TYPE ST_HMI_Machine :
STRUCT
	Command: ST_HMI_Machine_Command;
	Config: ST_HMI_Machine_Config;
	Status: ST_HMI_Machine_Status;
END_STRUCT
END_TYPE

(* stored: Version 1.1.0.1, ProductVersion 3.1.4024.12
   DUT ST_HMI_Machine: Id {cad70a19-def3-4322-83e5-729eb37116fe} *)
